// Brief: setup arm gravity calibration
// For trajectory synchronizaiton, the planner generate a trajecotry for setup joint3/5 and slave joint 1-3, but only former used here 
FUNCTION_BLOCK PUBLIC FB_SetupCtrlJnt5GraCali EXTENDS FB_SetupArmCtrlBase
VAR_INPUT
END_VAR
VAR_OUTPUT
END_VAR
VAR
// cali trajectory
	m_caliMotionSegs :INT :=3;
	m_graCaliTraj:ARRAY [1..3] OF LREAL:=[PI/2-pi/3, PI/2-PI/6, PI/2-pi/3];
	
		 
	m_caliMaxjntVel:LREAL:=2.5 * g_deg2Rad;
	m_caliMaxjntAcc:LREAL:=0.5;
	m_caliMaxjntJerk:LREAL:=2.0;
	
	m_caliTrajIdx: INT := 1;
	m_caliPlanner: ARRAY[1..3] OF FB_BasicDoubleS;
	
END_VAR

// override this function in each exact controller
METHOD PROTECTED calcCmdJntPos : BOOL
VAR_IN_OUT CONSTANT
	i_setupArm	:FB_SetupArm;
END_VAR


VAR 
	i :INT;
	curJntVel :Vec5d;
END_VAR
IF ABS(i_setupArm.curJntVel[5]) > 0.1 THEN
	m_isFinished:=TRUE;
	RETURN;
END_IF
// check if planner is ready
IF m_caliPlanner[m_caliTrajIdx].isGene = FALSE THEN
	calcCmdJntPos:=FALSE;
	RETURN;
END_IF

// traj plan
calcCmdJntPos :=m_caliPlanner[m_caliTrajIdx].evaluate(m_timePeriod, q=> m_cmdJntPos[5], q_dot=>m_cmdJntVel[5], q_ddot=> m_cmdJntAcc[5]);

// check if to transit to next segment
IF(m_timePeriod > m_caliPlanner[m_caliTrajIdx].duration  AND ABS(i_setupArm.curJntVel[5])<GVL_SlaveControlParameters.g_jntStaticVelThres) THEN
	m_caliTrajIdx:=m_caliTrajIdx+1;
	m_timePeriod:=0;
END_IF

// check if to terminated
IF(m_caliTrajIdx > m_caliMotionSegs) THEN
	m_isFinished:=TRUE;
END_IF
END_METHOD

METHOD PUBLIC init : BOOL
VAR_IN_OUT CONSTANT
	i_setupArm	:FB_SetupArm;
END_VAR
VAR_IN_OUT 
	r_setupArmCtrlCmd :ST_SetupArmCtrlCmds;
END_VAR

VAR
	i,j :INT;
	startJntPos,endJntPos :LREAL;
	q,v:ARRAY[1..2] OF lreal;
END_VAR
SUPER^.Init(i_setupArm,r_setupArmCtrlCmd);
m_jntEnableFlag[5]:=1;
m_caliTrajIdx :=1;

// traj plan
// fisrt segment
q[1]:=i_setupArm.curJntPos[5];
q[2]:=m_graCaliTraj[1];
v[1]:=0;
v[2]:=0;
m_caliPlanner[1].init(q,v,m_caliMaxjntVel, m_caliMaxJntAcc, m_caliMaxJntJerk);

// other segments
FOR i:=2 TO m_caliMotionSegs DO 
	q[1]:=m_graCaliTraj[i-1];
	q[2]:=m_graCaliTraj[i];
	m_caliPlanner[i].init(q,v,m_caliMaxjntVel, m_caliMaxJntAcc, m_caliMaxJntJerk);
END_FOR
END_METHOD

END_FUNCTION_BLOCK

(* stored: Version 1.1.0.1, ProductVersion 3.1.4024.11
   POU FB_SetupCtrlJnt5GraCali: Id {742a7c37-2108-447e-a095-ea9ab3206b7a}, SpecialFunc None
   Method calcCmdJntPos: Id {30706fea-fa22-4600-affa-2edaaea78691}
   Method init: Id {2e96f170-5dad-491c-ad85-3dab2234e4af} *)
